// TwinCAT 3 PLC project RED_PLC
// ProgramVersion: 3.1.4022.7
// libraries:
//   VisuElemBase, * (System)
//   Tc2_Standard, * (Beckhoff Automation GmbH)
//   Tc2_System, * (Beckhoff Automation GmbH)
//   Tc3_Module, * (Beckhoff Automation GmbH)
//   VisuDialogs, * (System)
//   Mercury ,0.0.0.60,Johnson Matthey Technology Centre
//   VisuSymbols,3.5.10.0,System
// project tree:
//   DUTs/DATATYPES/ _ST_DATA_.TcDUT, _ST_ERROR_.TcDUT
//   DUTs/HMI/ _ST_BLANK_2_.TcDUT, _ST_BLANK_1_.TcDUT, _ST_HOME_.TcDUT, _ST_SETTINGS_.TcDUT
//   DUTs/IO/ _ST_EL1008_M11_.TcDUT, _ST_EL1008_M12_.TcDUT, _ST_EL2008_M13_.TcDUT, _ST_MKS_MFC_.TcDUT
//   / GlobalTextList.TcGTLO, PlcTask.TcTTO, HgV_Task.TcTTO, VISU_TASK.TcTTO
//   GVLs/ CONSTANTS.TcGVL, HMI.TcGVL, IO.TcGVL, PC.TcGVL
//   POUs/00_Application/ MAIN.TcPOU
//   POUs/01_System/ FB_Beckhoff_EV.TcPOU
//   POUs/02_Subsystems/ FB_Beckhoff_Electric_Propulsion.TcPOU, FB_Beckhoff_Auxilary.TcPOU, FB_Beckhoff_Energy_Source.TcPOU
//   VISUs/00_Front_Page/ FP.TcVIS, Navigation_Bar.TcVIS
//   VISUs/01_Pages/ _000_Home.TcVIS, _001_Blank_1.TcVIS, _002_Blank_2.TcVIS, _003_Settings.TcVIS
//   VISUs/98_Visualization Manager/ VisualizationManager.TcVMO (not stored)

CONFIGURATION RED_PLC
    RESOURCE PLC ON TwinCAT3
        TASK PlcTask(INTERVAL := T#10ms, PRIORITY := 20);
        TASK HgV_Task(INTERVAL := T#10ms, PRIORITY := 1);
        TASK VISU_TASK(INTERVAL := T#200000us, PRIORITY := 30);
        PROGRAM MAIN WITH PlcTask : MAIN;
        PROGRAM HgV_Engine WITH HgV_Task : HgV_Engine;
        PROGRAM VisuElems_Visu_Prg WITH VISU_TASK : VisuElems.Visu_Prg;
    END_RESOURCE
END_CONFIGURATION

// ---- DUTs/DATATYPES/_ST_DATA_.TcDUT
 TYPE _ST_DATA_ :
STRUCT
END_STRUCT
END_TYPE

// ---- DUTs/DATATYPES/_ST_ERROR_.TcDUT
TYPE _ST_ERROR_ :
STRUCT
	CODE 	: INT;
	SOURCE 	: STRING(255);
	STATUS 	: BOOL;
END_STRUCT
END_TYPE

// ---- DUTs/HMI/_ST_BLANK_2_.TcDUT
TYPE _ST_BLANK_2_ :
STRUCT
END_STRUCT
END_TYPE

// ---- DUTs/HMI/_ST_BLANK_1_.TcDUT
TYPE _ST_BLANK_1_ :
STRUCT
END_STRUCT
END_TYPE

// ---- DUTs/HMI/_ST_HOME_.TcDUT
TYPE _ST_HOME_ :
STRUCT
END_STRUCT
END_TYPE

// ---- DUTs/HMI/_ST_SETTINGS_.TcDUT
TYPE _ST_SETTINGS_ :
STRUCT
END_STRUCT
END_TYPE

// ---- DUTs/IO/_ST_EL1008_M11_.TcDUT
// EL1008 | 8-channel digital input terminal 24 V DC, 3 ms
// NAMING CONVENTION: bCHX_XXXXX... e.g bCH1_EXTRACT_ALARM
TYPE _ST_EL1008_M11_ :
STRUCT
	bCH1 AT %I* : BOOL;
	bCH2 AT %I*	: BOOL;
	bCH3 AT %I*	: BOOL;
	bCH4 AT %I*	: BOOL;
	bCH5 AT %I*	: BOOL;
	bCH6 AT %I*	: BOOL;
	bCH7 AT %I*	: BOOL;
	bCH8 AT %I*	: BOOL;
END_STRUCT
END_TYPE

// ---- DUTs/IO/_ST_EL1008_M12_.TcDUT
// EL1008 | 8-channel digital input terminal 24 V DC, 3 ms
// NAMING CONVENTION: bCHX_XXXXX... e.g bCH1_EXTRACT_ALARM
TYPE _ST_EL1008_M12_ :
STRUCT
	bCH1 AT %I* : BOOL;
	bCH2 AT %I*	: BOOL;
	bCH3 AT %I*	: BOOL;
	bCH4 AT %I*	: BOOL;
	bCH5 AT %I*	: BOOL;
	bCH6 AT %I*	: BOOL;
	bCH7 AT %I*	: BOOL;
	bCH8 AT %I*	: BOOL;
END_STRUCT
END_TYPE

// ---- DUTs/IO/_ST_EL2008_M13_.TcDUT
// EL2008 | 8-channel digital output terminal 24 V DC, 0.5 A
// NAMING CONVENTION: bCHX_XXXXX... e.g bCH1_EXTRACT_ALARM
TYPE _ST_EL2008_M13_ :
STRUCT
	bCH1 AT %Q* : BOOL;
	bCH2 AT %Q*	: BOOL;
	bCH3 AT %Q*	: BOOL;
	bCH4 AT %Q*	: BOOL;
	bCH5 AT %Q*	: BOOL;
	bCH6 AT %Q*	: BOOL;
	bCH7 AT %Q*	: BOOL;
	bCH8 AT %Q*	: BOOL;
END_STRUCT
END_TYPE

// ---- DUTs/IO/_ST_MKS_MFC_.TcDUT
TYPE _ST_MKS_MFC_ :
STRUCT
	iEXCEPTION_STATUS	AT %I*	: USINT;
	fFLOW_READING		AT %I*	: REAL;
	fACTUATOR_CURRENT	AT %I*	: REAL;
	
	fFLOW_SP 			AT %Q*	: REAL;
	iACTUATOR_CONTROL	AT %Q*	: USINT;
	iRAMP_TIME			AT %Q*	: UDINT;
END_STRUCT
END_TYPE

// ---- GVLs/CONSTANTS.TcGVL
{attribute 'qualified_only'}
VAR_GLOBAL CONSTANT
	iNUMBER_OF_MFC : INT := 2; // Maximum number of MFC's in system
END_VAR

// ---- GVLs/HMI.TcGVL
//HMI Pages/Variables here. RETAIN PERSISTANT variables must be declares at the top.
VAR_GLOBAL RETAIN PERSISTENT
	SETTINGS	: _ST_SETTINGS_;
END_VAR
VAR_GLOBAL
	HOME 		: _ST_HOME_;
	BLANK_1 	: _ST_BLANK_1_;
	BLANK_2 	: _ST_BLANK_2_;
END_VAR

// ---- GVLs/IO.TcGVL
// IO Structures/Variables. Avoid declaring IO in PROGRAMS FUNCTIONS and FUNCTION BLOCKS
VAR_GLOBAL
		stEL1008_M11 	: _ST_EL1008_M11_;
		stEL1008_M12 	: _ST_EL1008_M11_;
		stEL1008_M13 	: _ST_EL1008_M11_;
		stMFC 			: ARRAY[1..CONSTANTS.iNUMBER_OF_MFC] OF _ST_MKS_MFC_;
END_VAR

// ---- GVLs/PC.TcGVL
// Variables to be accessed by Labview or PC.
VAR_GLOBAL
END_VAR

// ---- POUs/00_Application/MAIN.TcPOU
PROGRAM MAIN
VAR
	fbCar 	: FB_Beckhoff_EV;
END_VAR

fbCar();

END_PROGRAM

// ---- POUs/01_System/FB_Beckhoff_EV.TcPOU
FUNCTION_BLOCK FB_Beckhoff_EV
VAR_INPUT
END_VAR
VAR_OUTPUT
END_VAR
VAR
END_VAR

END_FUNCTION_BLOCK

// ---- POUs/02_Subsystems/FB_Beckhoff_Electric_Propulsion.TcPOU
FUNCTION_BLOCK FB_Beckhoff_Electric_Propulsion
VAR_INPUT
END_VAR
VAR_OUTPUT
END_VAR
VAR
END_VAR

END_FUNCTION_BLOCK

// ---- POUs/02_Subsystems/FB_Beckhoff_Auxilary.TcPOU
FUNCTION_BLOCK FB_Beckhoff_Auxilary
VAR_INPUT
END_VAR
VAR_OUTPUT
END_VAR
VAR
END_VAR

END_FUNCTION_BLOCK

// ---- POUs/02_Subsystems/FB_Beckhoff_Energy_Source.TcPOU
FUNCTION_BLOCK FB_Beckhoff_Energy_Source
VAR_INPUT
END_VAR
VAR_OUTPUT
END_VAR
VAR
END_VAR

END_FUNCTION_BLOCK

// ---- GlobalTextList.TcGTLO
TEXTLIST GlobalTextList
  18 = '%.2f Bar'
  660 = '%.3f slpm'
  647 = '%02d'
  649 = '%s'
  21 = '%t[HH : mm : ss]'
  24 = '%t[HH:mm :ss]'
  676 = 'Admin'
  175 = 'ARCHIVED SEQUENCES'
  80 = 'BLANK 1'
  392 = 'BLANK 2'
  173 = 'BUILD SEQUENCE'
  6 = 'CANCEL'
  797 = 'DEFAULT'
  645 = 'DONE'
  659 = 'FLOW RATE'
  604 = 'FLOW RATE THRESHOLDS'
  603 = 'GAS MIX'
  22 = 'GAS MIX PRESSURE'
  243 = 'Gas Supply'
  648 = 'HH'
  172 = 'HOME'
  590 = 'LOGIN'
  231 = 'LOGOUT'
  4 = 'MM'
  961 = 'N2O2 MIX PRESSURE'
  25 = 'NITROGEN'
  965 = 'Nitrogen Channel Status'
  607 = 'NITROGEN FLOW RATE'
  962 = 'NITROGEN PRESSURE'
  697 = 'None'
  143 = 'Operator'
  658 = 'OXYGEN'
  964 = 'Oxygen Channel Status'
  606 = 'OXYGEN FLOW RATE'
  608 = 'OXYGEN PRESSURE '
  17 = 'PRESSURE'
  602 = 'PRESSURE THRESHOLDS'
  798 = 'RESET ERROR'
  26 = 'SEQUENCE'
  589 = 'Service'
  244 = 'Set System Thresholds'
  174 = 'SETTINGS'
  5 = 'SS'
  19 = 'SYSTEM'
  605 = 'System Readings'
  963 = 'System Status'
  20 = 'TIME ELAPSED'
  646 = 'Time Picker'
  23 = 'TOTAL TIME'
  316 = 'WIDGET 1'
  85 = 'WIDGET 2'
  637 = 'WIDGET 3'
END_TEXTLIST

// ---- VISUs/00_Front_Page/FP.TcVIS
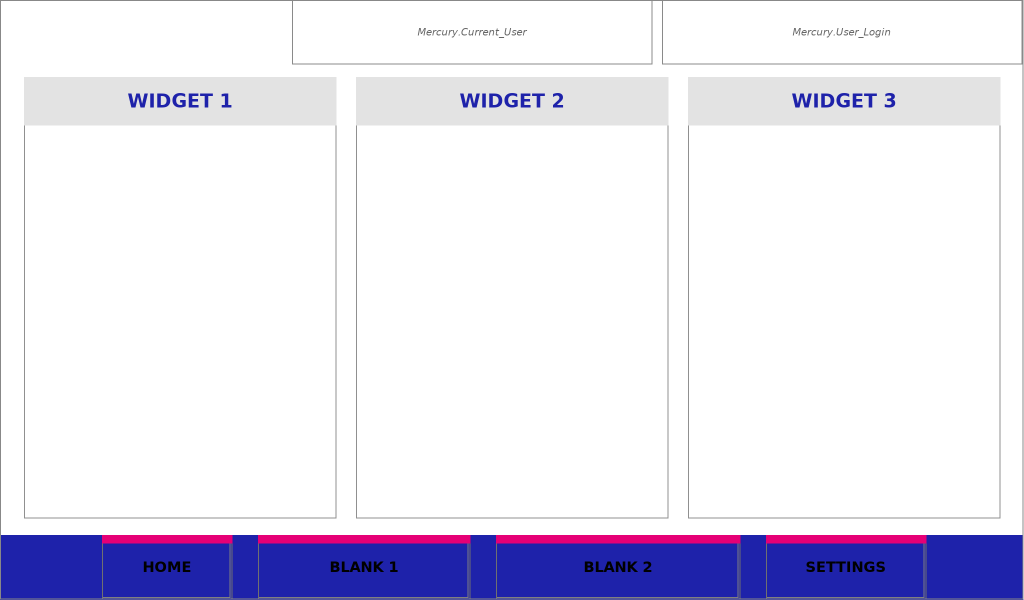
VISUALIZATION FP  // 1024x600, background image JMTC.Swindon_Glovebox_UI_Background
    Frame (0,535 1023x65)
        shows Navigation_Bar()
    Frame (292,0 360x64)
        shows Mercury.Current_User()
    Frame (662,0 360x64), invisible if: HgV_Engine.stNav_Button[3].bInvisible
        shows Mercury.User_Login()
    Frame (0,60 1024x472), frame switch variable: HgV_Engine.propCurrent_Page_
        shows _000_Home()
        shows _001_Blank_1()
        shows _002_Blank_2()
        shows _003_Settings()
END_VISUALIZATION

// ---- VISUs/00_Front_Page/Navigation_Bar.TcVIS
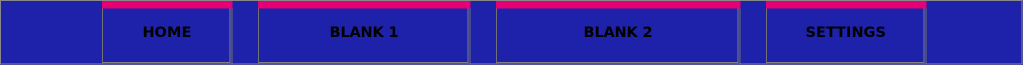
VISUALIZATION Navigation_Bar  // 1023x65
    Button (102,0 130x64), "HOME", image: JMTC.JMTC_Home_icon_32px
        tap HgV_Engine.stNav_Button[0].bToggle
    Button (258,0 212x64), "BLANK 1", image: JMTC.jmtc_sequence_icon_32px
        tap HgV_Engine.stNav_Button[1].bToggle
    Button (766,0 160x64), "SETTINGS", image: JMTC.jmtc_config_icon_32px
        tap HgV_Engine.stNav_Button[3].bToggle
    Rectangle (258,0 212x8), invisible if: HgV_Engine.stNav_Button[1].bInvisible
    Button (496,0 244x64), "BLANK 2", image: JMTC.jmtc_archive2_icon_32px
        tap HgV_Engine.stNav_Button[2].bToggle
    Rectangle (102,0 130x8), invisible if: HgV_Engine.stNav_Button[0].bInvisible
    Rectangle (496,0 244x8), invisible if: HgV_Engine.stNav_Button[2].bInvisible
    Rectangle (766,0 160x8), invisible if: HgV_Engine.stNav_Button[3].bInvisible
END_VISUALIZATION

// ---- VISUs/01_Pages/_000_Home.TcVIS
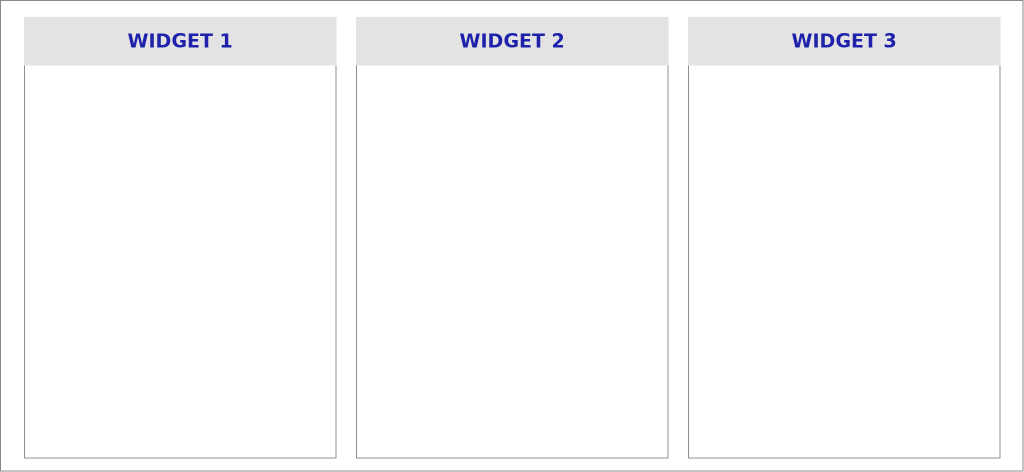
VISUALIZATION _000_Home  // 1024x472
    GroupBox (24,16 312x442)
        Rectangle (0,1 312x48), "WIDGET 1"
    GroupBox (356,16 312x442)
        Rectangle (0,1 312x48), "WIDGET 2"
    GroupBox (688,16 312x442)
        Rectangle (0,1 312x48), "WIDGET 3"
END_VISUALIZATION

// ---- VISUs/01_Pages/_001_Blank_1.TcVIS
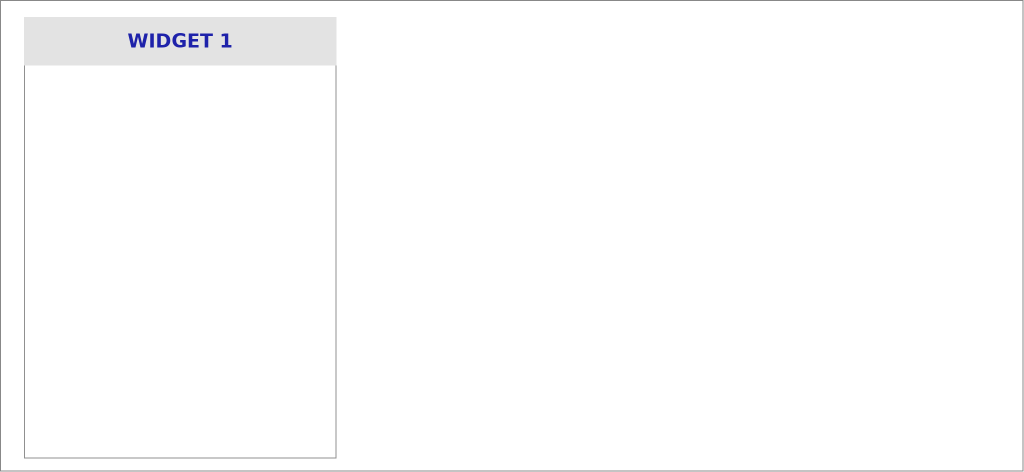
VISUALIZATION _001_Blank_1  // 1024x472
    GroupBox (24,16 312x442)
        Rectangle (0,1 312x48), "WIDGET 1"
END_VISUALIZATION

// ---- VISUs/01_Pages/_002_Blank_2.TcVIS
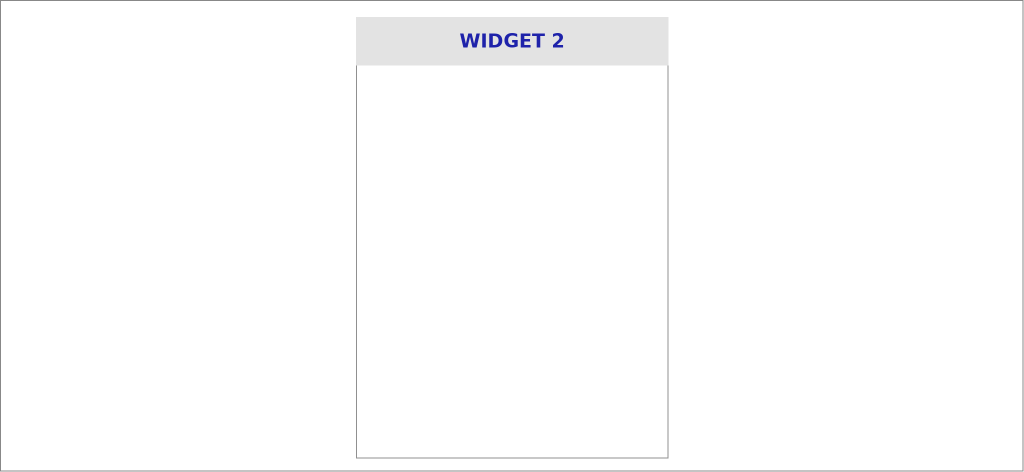
VISUALIZATION _002_Blank_2  // 1024x472
    GroupBox (356,16 312x442)
        Rectangle (0,1 312x48), "WIDGET 2"
END_VISUALIZATION

// ---- VISUs/01_Pages/_003_Settings.TcVIS
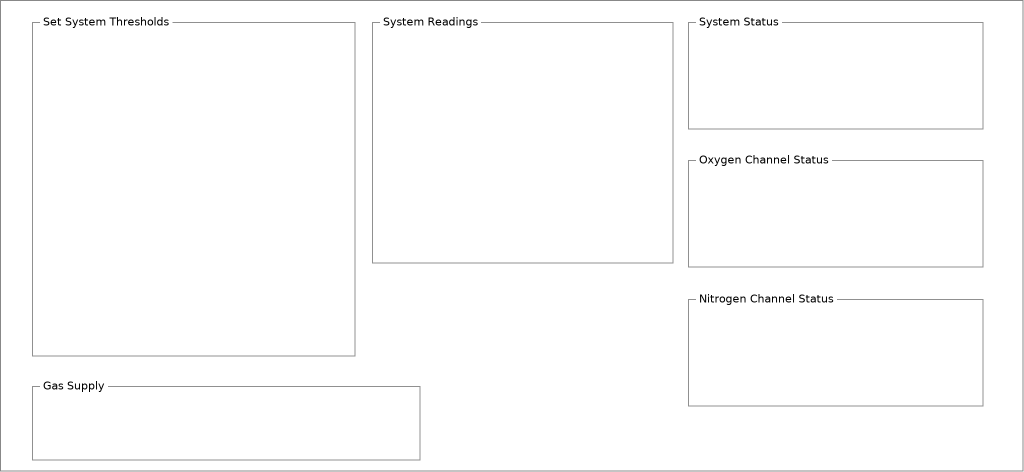
VISUALIZATION _003_Settings  // 1024x472
    GroupBox (32,378 388x82), "Gas Supply"
    GroupBox (32,14 323x342), "Set System Thresholds"
    GroupBox (372,14 301x249), "System Readings"
    GroupBox (688,14 295x115), "System Status"
    GroupBox (688,152 295x115), "Oxygen Channel Status"
    GroupBox (688,291 295x115), "Nitrogen Channel Status"
END_VISUALIZATION
